// TIA Portal V20 export
DATA_BLOCK "Diag_DB"   // DB60
// stored: AutoNumber false, InstanceOfName Diag, InstanceOfType FB
"Diag"
   // VAR
   //    Var { ExternalAccessible := 'False'; ExternalVisible := 'False'; ExternalWritable := 'False'} : "TypeVar";
   //    Plc { ExternalAccessible := 'False'; ExternalVisible := 'False'; ExternalWritable := 'False'} : "Diag_PLCCheck";
   //    PlcData { ExternalAccessible := 'False'; ExternalVisible := 'False'; ExternalWritable := 'False'} : "UserDiag_typePLC";
   //    IoSys1 { ExternalAccessible := 'False'; ExternalVisible := 'False'; ExternalWritable := 'False'} : "Diag_IOSystemCheck";
   //    IoDataSys1 { ExternalAccessible := 'False'; ExternalVisible := 'False'; ExternalWritable := 'False'} : "UserDiag_typeIOSystem";
   // END_VAR
BEGIN
END_DATA_BLOCK
